// Mitsubishi GX Works2 project: 23   PLC: FX3G

// task Task_01 (event TRUE, interval 0, priority 31): POU_01

PROGRAM POU_01
VAR
  wstep : INT;
  ton1 : TON;
END_VAR
M99 := FALSE AND
M1 AND
Y0 AND Y1 AND Y2 AND Y3;

IF M8002 THEN
	wstep := 0;
END_IF;

CASE wstep OF
	0:
		zrst(TRUE, Y0, Y100);
		ton1(in := FALSE);
	
		IF M1 THEN
			wstep := 20;
		END_IF;
		
	20:
		Y0 := TRUE;
		Y1 := TRUE;
		ton1(in := NOT ton1.q, pt := t#5s);
	
		IF NOT M1 THEN
			wstep := 0;
		END_IF;
		IF ton1.q THEN
			wstep := 21;
		END_IF;
	21:
		Y2 := TRUE;
		ton1(in := NOT ton1.q, pt := t#10s);
		
		IF NOT M1 THEN
			wstep := 0;
		END_IF;
		IF ton1.q THEN
			wstep := 22;
		END_IF;
	22:
		Y3 := TRUE;
		
		IF NOT M1 THEN
			wstep := 0;
		END_IF;
END_CASE;
END_PROGRAM
